TYPE enum_E:
    (elit_l1, elit_l10, elit_l11, elit_l12, elit_l13, elit_l14, elit_l15, elit_l16, elit_l2, elit_l3, elit_l4, elit_l5, elit_l6, elit_l7, elit_l8, elit_l9, elit_LIT1, elit_LIT2);
END_TYPE

(* stored: ProductVersion 3.1.0.18, Version 1.1.0.1 *)
